(* IEC 61131-3 sources: test/Class/Sfc_Action_Base, 1 file *)

(* ---- Sfc_Action_Base.st ---- *)
(*!
<Class
	Name               = "Sfc_Action_Base"
	Revision           = "2.0"
	RealtimeTask       = "false"
	CyclicTask         = "false"
	BackgroundTask     = "false"
	Sigmatek           = "true"
	OSInterface        = "false"
	HighPriority       = "false"
	Automatic          = "false"
	UpdateMode         = "Prescan"
	SharedCommandTable = "true"
	Objectsize         = "(284,120)">
	<Channels>
		<Server Name="A" Visualized="true" Initialize="false" WriteProtected="true" Retentive="false" Comment="Active flag&#13;&#10;&#13;&#10;Indicates if the action is active"/>
		<Server Name="DelayActive" Visualized="false" Initialize="false" WriteProtected="true" Retentive="false" Comment="Delay flag&#13;&#10;&#13;&#10;Indicates that the action is&#13;&#10;waiting for a time delay in order&#13;&#10;to become active"/>
		<Server Name="Itf" Visualized="false" Initialize="false" WriteProtected="true" Retentive="false" Comment="Interface to the action class"/>
		<Server Name="Q" Visualized="true" Initialize="false" WriteProtected="true" Retentive="false" Comment="Last execution flag&#13;&#10;&#13;&#10;Indicates that the action has become&#13;&#10;inactive and is being executed for the last time."/>
		<Server Name="T" Visualized="true" Initialize="false" WriteProtected="true" Retentive="false" Comment="Action timer&#13;&#10;&#13;&#10;If the action is active, the value&#13;&#10;of the action timer is the time since&#13;&#10;the activation of the action.&#13;&#10;Otherwise the value of the action timer&#13;&#10;is the duration of the last active phase.&#13;&#10;&#13;&#10;Unit: ms"/>
		<Client Name="GetParentPtr" Required="true" Internal="false" Comment="Helper client for optaining a&#13;&#10;pointer to the parent SFC class."/>
		<Client Name="LogonToInvoker" Required="true" Internal="false" Comment="Helper Client for registration&#13;&#10;at the action invoker."/>
	</Channels>
	<RevDoku>
		<Owner Company="Sigmatek GmbH &amp; Co KG" Author="LesMax"/>
		<Dokumentation Revision="2.0" Date="2014-05-20" Author="LesMax" Company="Sigmatek GmbH &amp; Co KG" Description="Introduced new action priority management&#13;&#10;for a defined calling sequence."/>
		<Dokumentation Revision="1.2" Date="2013-12-04" Author="LesMax" Company="Sigmatek GmbH &amp; Co KG" Description="The Servers &quot;DelayActive&quot; and &quot;AtRisingEdge&quot; are now always reset at the beginning of the &quot;OnStepActive&quot; Method."/>
		<Dokumentation Revision="1.1" Date="2013-10-17" Author="LesMax" Company="Sigmatek GmbH &amp; Co KG" Description="Actions now obtain a pointer to the&#13;&#10;parent Sfc class at initialisation."/>
	</RevDoku>
	<Network Name="Sfc_Action_Base">
		<!-- List of Components in this network -->
		<Components>
		</Components>
		<Comments>
		</Comments>
		<!-- List of Connections in this network -->
		<Connections>
		</Connections>
		<!-- Headerfiles -->
		<Options>
		</Options>
	</Network>
</Class>
*)
Sfc_Action_Base : CLASS
	TYPE
	  ActionQualifiers :  //! <Type Public="true" Name="ActionQualifiers"/>
	  (
	    N_Qualifier,
	    R_Qualifier,
	    S_Qualifier,
	    L_Qualifier,
	    D_Qualifier,
	    P_Qualifier,
	    P0_Qualifier,
	    P1_Qualifier,
	    SD_Qualifier,
	    DS_Qualifier,
	    SL_Qualifier
	  )$UDINT;
	  PriorityOffset :
	  (
	    OffsetAtRisingEdge:=0,
	    OffsetRegular:=150000,
	    OffsetAtFallingEdge:=300000
	  )$UDINT;
	  PtrTo_Sfc_Network_Base : ^Sfc_Network_Base;
	END_TYPE
  //Servers:
	Itf 	: SvrChCmd_DINT;
	A 	: SvrCh_DINT;
	T 	: SvrCh_UDINT;
	Q 	: SvrCh_DINT;
	DelayActive 	: SvrCh_DINT;
  //Clients:
	LogonToInvoker 	: CltCh_pVoid;
	GetParentPtr 	: CltCh_UDINT;
  //Variables:
		m_ActionQualifier 	: ActionQualifiers;			//! <Variable Comment="Action qualifier&#13;&#10;&#13;&#10;Currently used action qualifier" Name="m_ActionQualifier"/>
		m_TimerSetting 	: UDINT;			//! <Variable Comment="Time setting&#13;&#10;&#13;&#10;Optional time setting for limited or delayed actions" Name="m_TimerSetting"/>
		m_Priority 	: UDINT;
		m_ActiveTimeStamp 	: UDINT;			//! <Variable Comment="Time stamp&#13;&#10;&#13;&#10;Time stamp for active phase duration measuring" Name="m_ActiveTimeStamp"/>
		m_DelayTimeStamp 	: UDINT;			//! <Variable Comment="Delay time stamp&#13;&#10;&#13;&#10;Time stamp for time delayed actions" Name="m_DelayTimeStamp"/>
  //Functions:

	FUNCTION Sfc_Action_Base
		VAR_OUTPUT
			ret_code 	: ConfStates;
		END_VAR;

	FUNCTION VIRTUAL GLOBAL Init;

	FUNCTION VIRTUAL GLOBAL Work;

	FUNCTION VIRTUAL GLOBAL LastWorkPass;

	FUNCTION DoWork;

	FUNCTION VIRTUAL OnWork;

	FUNCTION VIRTUAL OnActive;

	FUNCTION VIRTUAL OnInactive;

	FUNCTION DoActive;

	FUNCTION DoInactive;

	FUNCTION CalculateDelayTime
		VAR_OUTPUT
			DelayTime 	: UDINT;
		END_VAR;

	FUNCTION CalculateActiveTime
		VAR_OUTPUT
			ActiveTime 	: UDINT;
		END_VAR;

	FUNCTION HandleTimeLimit;

	FUNCTION HandlePulse;

	FUNCTION GLOBAL OnStepActive
		VAR_INPUT
			ActionQualifier 	: ActionQualifiers;
			TimerSetting 	: UDINT;
		END_VAR;

	FUNCTION GLOBAL OnStepInactive;

	FUNCTION GLOBAL HandleTimeDelay;

	FUNCTION VIRTUAL OnReadInternalVariables;

	FUNCTION VIRTUAL OnWriteInternalVariables;

	FUNCTION GLOBAL SetPriority
		VAR_INPUT
			Priority 	: UDINT;
		END_VAR;

	FUNCTION GLOBAL GetPriority
		VAR_OUTPUT
			Priority 	: UDINT;
		END_VAR;

	FUNCTION GLOBAL UpdatePriorities;
  //Tables:
	FUNCTION @STD
		VAR_OUTPUT
			ret_code	: CONFSTATES;
		END_VAR;
	FUNCTION GLOBAL TAB @CT_;
END_CLASS;

#pragma usingLtd Sfc_Network_Base

// Init method for registering at action invoker
FUNCTION VIRTUAL GLOBAL Sfc_Action_Base::Init

  if _FirstScan then

    LogonToInvoker.Write(input:=this);

    GetParentPtr := GetParentPtr.Read();

  end_if;

END_FUNCTION

// Implement Worker Interface
FUNCTION VIRTUAL GLOBAL Sfc_Action_Base::Work

  // Call own work routine if active
  if A = 1 then

    // Read all connected internal variable servers
    OnReadInternalVariables();

    // Call work routine
    DoWork();

    // Write all connected internal variable servers
    OnWriteInternalVariables();

    // Handle the limited action qualifiers
    HandleTimeLimit();

    // Handle the pulse action qualifiers
    HandlePulse();

  end_if;

END_FUNCTION

// Handles actions wich were deactivated in the last cycle
// as well as actions that are called at a falling edge
FUNCTION VIRTUAL GLOBAL Sfc_Action_Base::LastWorkPass

  if A = 0 & Q = 1 then

    // Read all connected internal variable servers
    OnReadInternalVariables();

    // Call work routine one last time
    DoWork();

    // Write all connected internal variable servers
    OnWriteInternalVariables();

    // Reset Q flag
    Q := 0;

    DoInactive();

  end_if;

END_FUNCTION

FUNCTION Sfc_Action_Base::DoWork

  // Update the execution timer
  T := CalculateActiveTime();

  // Call User Work Handler
  OnWork();

END_FUNCTION

FUNCTION Sfc_Action_Base::DoActive

  // Save a timestamp for the activation of the action
  m_ActiveTimeStamp := ops.tAbsolute;

  // Reset the execution timer
  T := 0;

  // Call User active Handler
  OnActive();

END_FUNCTION

FUNCTION Sfc_Action_Base::DoInactive

  // Reset the activation timestamp
  m_ActiveTimeStamp := 0;

  // Call User Inactive Handler
  OnInactive();

END_FUNCTION

FUNCTION Sfc_Action_Base::CalculateDelayTime
	VAR_OUTPUT
		DelayTime 	: UDINT;
	END_VAR
    VAR
    curTime : UDINT;
  END_VAR

    // Calculate delay time
    curTime := ops.tAbsolute;

    // Handle Overflow condition
    if curTime < m_DelayTimeStamp then

      DelayTime := curTime + sizeof(UDINT) - m_DelayTimeStamp;

    else

      DelayTime := curTime - m_DelayTimeStamp;

    end_if;

END_FUNCTION

FUNCTION Sfc_Action_Base::CalculateActiveTime
	VAR_OUTPUT
		ActiveTime 	: UDINT;
	END_VAR
  VAR
  	curTime : UDINT;
  END_VAR

  // Update the execution timer
  curTime := ops.tAbsolute;

  // Handle Overflow condition
  if curTime < m_ActiveTimeStamp then

    ActiveTime := curTime + sizeof(UDINT) - m_ActiveTimeStamp;

  else

    ActiveTime := curTime - m_ActiveTimeStamp;

  end_if;

END_FUNCTION

FUNCTION Sfc_Action_Base::HandleTimeLimit

  case m_ActionQualifier of

  L_Qualifier, SL_Qualifier:

    // Check if the time limit is reached
    if CalculateActiveTime() >= m_TimerSetting then

      A := 0;
      Q := 1;

    end_if;

  end_case;

END_FUNCTION

FUNCTION Sfc_Action_Base::HandlePulse

  case m_ActionQualifier of

  P_Qualifier, P1_Qualifier:

    A := 0;
    Q := 0;

  end_case;

END_FUNCTION

FUNCTION GLOBAL Sfc_Action_Base::HandleTimeDelay

  case m_ActionQualifier of

  D_Qualifier, DS_Qualifier, SD_Qualifier:

    if DelayActive = 1 & CalculateDelayTime() >= m_TimerSetting then

      A := 1;
      Q := 0;

      m_DelayTimeStamp := 0;
      DelayActive := 0;

      DoActive();

    end_if;

  end_case;

END_FUNCTION

FUNCTION GLOBAL Sfc_Action_Base::OnStepActive
	VAR_INPUT
		ActionQualifier 	: ActionQualifiers;
		TimerSetting 	: UDINT;
	END_VAR

  m_ActionQualifier := ActionQualifier;
  m_TimerSetting := TimerSetting;
  DelayActive := 0;

  case m_ActionQualifier of

  R_Qualifier:

    A := 0;
    Q := 1;

  D_Qualifier, SD_Qualifier, DS_Qualifier:

    A := 0;
    Q := 0;

    m_DelayTimeStamp := ops.tAbsolute;
    DelayActive := 1;

  P0_Qualifier:

    A := 0;
    Q := 0;

  P_Qualifier, P1_Qualifier:

    A := 1;
    Q := 0;

    DoActive();

  else

    A := 1;
    Q := 0;

    DoActive();

  end_case;

END_FUNCTION

FUNCTION GLOBAL Sfc_Action_Base::OnStepInactive

  case m_ActionQualifier of

  N_Qualifier, L_Qualifier, D_Qualifier:

    if A = 1 then

      A := 0;
      Q := 1;

    end_if;

    m_DelayTimeStamp := 0;
    DelayActive := 0;

  P_Qualifier, P0_Qualifier:

    A := 0;
    Q := 1;

    m_DelayTimeStamp := 0;
    DelayActive := 0;

  SD_Qualifier:

    // Do nothing (leave the delay timer active)

  else

    m_DelayTimeStamp := 0;
    DelayActive := 0;

  end_case;

END_FUNCTION

// Constructor
FUNCTION Sfc_Action_Base::Sfc_Action_Base
	VAR_OUTPUT
		ret_code 	: ConfStates;
	END_VAR

  m_ActionQualifier     := N_Qualifier;
  m_Priority            := 0;
  m_TimerSetting        := 0;
  m_ActiveTimeStamp     := 0;
  m_DelayTimeStamp      := 0;

  ret_code := C_OK;

END_FUNCTION

// Overrideable for user work handler
FUNCTION VIRTUAL Sfc_Action_Base::OnWork

END_FUNCTION

// Overrideable for user activation handler
FUNCTION VIRTUAL Sfc_Action_Base::OnActive

END_FUNCTION

// Overrideable for user deactivation handler
FUNCTION VIRTUAL Sfc_Action_Base::OnInactive

END_FUNCTION

// Overrideable for reading connected internal variable servers
FUNCTION VIRTUAL Sfc_Action_Base::OnReadInternalVariables

END_FUNCTION

// Overrideable for writing connected internal variable servers
FUNCTION VIRTUAL Sfc_Action_Base::OnWriteInternalVariables

END_FUNCTION

FUNCTION GLOBAL Sfc_Action_Base::SetPriority
	VAR_INPUT
		Priority 	: UDINT;
	END_VAR

  m_Priority := Priority;

END_FUNCTION

FUNCTION GLOBAL Sfc_Action_Base::GetPriority
	VAR_OUTPUT
		Priority 	: UDINT;
	END_VAR

  case m_ActionQualifier of

  P_Qualifier:

    if (A = 0) & Q then

      Priority := m_Priority + OffsetAtFallingEdge$UDINT;

    else

      Priority := m_Priority + OffsetAtRisingEdge$UDINT;

    end_if;

  P0_Qualifier:

    Priority := m_Priority + OffsetAtFallingEdge$UDINT;

  P1_Qualifier:

    Priority := m_Priority + OffsetAtRisingEdge$UDINT;

  else

    Priority := m_Priority + OffsetRegular$UDINT;

  end_case;

END_FUNCTION

FUNCTION GLOBAL Sfc_Action_Base::UpdatePriorities

  if GetParentPtr <> NIL then

    GetParentPtr$PtrTo_Sfc_Network_Base^.UpdateActionPriorities();

  end_if;

END_FUNCTION
